Staubli VAL3: IsUseSameTool.pgx

public program IsUseSameTool(string& x_sCheck[], bool& x_bResult)
  local num i
  local string l_sEvent
  local tool l_tTool
  local tool l_tOldTool
begin
  l_tOldTool.trsf.x=-123456
  x_bResult=true
  for i=0 to size(x_sCheck)-1
    if left(x_sCheck[i],4)=="TRAJ"
      l_sEvent=right(x_sCheck[i],len(x_sCheck[i])-5)
      if isDefined(trajPt:tTraj[l_sEvent])
        // use the type...
        tTraies=trajPt:tTraj[l_sEvent]
      endIf
      call getTrajTool(l_tTool,tTraies.nIndexTool)

    endIf
    if left(x_sCheck[i],6)=="JPOINT"
      l_sEvent=right(x_sCheck[i],len(x_sCheck[i])-7)
      if isDefined(jPt:tTraj[l_sEvent])
        // use the type...
        tTrajJoint=jPt:tTraj[l_sEvent]
      endIf
      call getTrajTool(l_tTool,tTrajJoint.nIndexTool)
    endIf
    if l_tOldTool.trsf.x==-123456
      l_tOldTool=l_tTool
    else
      if l_tOldTool!=l_tTool
        x_bResult=false
        return
      endIf
    endIf
  endFor
end
